{attribute 'pack_mode' := '2'}
TYPE stKL306x_Channel:
STRUCT
	State 	AT %I* : stKL306x_ChannelStatus;	 
	DataIn 	AT %I* : INT;  
END_STRUCT
END_TYPE;

(* stored: Version 1.1.0.1, ProductVersion 3.1.4024.9
   DUT stKL306x_Channel: Id {a08c09fb-1429-486d-b2a3-d327c6899174} *)
